# B&R Automation Studio project NAELD004C00R10L518F00 (part 34)

#### Local.var
```iecst
(*2020-03-16*)
(**)
(*Local Action, State & Status*)
VAR
	eAct : eLifterAction := LifterActIdle;
	eStat : eLifterAction := LifterActIdle;
	eMainStatus : eFBStatus := Idle;
	eStatus : eFBStatus := Idle;
	eStatus1 : eFBStatus := Idle;
	eStatus2 : eFBStatus := Idle;
	eStatus3 : eFBStatus := Idle;
	udiStatus : UDINT := 0;
	udiStatus1 : UDINT := 0;
	udiStatus2 : UDINT := 0;
	udiStatus3 : UDINT := 0;
	sStatTxt : STRING[200] := '';
	a_sStatText : ARRAY[0..50] OF STRING[200] := ['Idling','Going A Position','Going B Position','Going C Position','Going D Position','Going E Position','Going F Position','Going G Position','Going H Position','Going A Slot Position','Going Next A Slot Position','Going Previous A Slot Position','Going B Slot Position','Going Next B Slot Position','Going Previous B Slot Position','Going C Slot Position','Going Next C Slot Position','Going Previous C Slot Position','Going D Slot Position','Going Next D Slot Position','Going Previous D Slot Position','Full Homing','Powering On','Powering Off','Homing','Moving Absolute','Moving Relative','Jogging Up','Jogging Down','Jogging Stop','Resetting Axis Error','Stopping','Writing SDO','Background Starting Module OK Check','Background Stopping Module OK Check','Full Moving Relative','Reset Servo Module Node',14('')];
END_VAR
(**)
(*Local Alarm*)
VAR
	tyAlmData : tyAlmDat;
	tyAlmData1 : tyAlmDat;
	tyAlmData2 : tyAlmDat;
	tyAlmData3 : tyAlmDat;
	a_tyAlmText : ARRAY[10000..10299] OF tyAlmTxt := [(sAlmText:='Axis Move Abnormally By External Force',sRcyText:='Servo Motor Abnormal Operation. Reset And Resume Operation. If The Problem Persists, Please Contact Nutek For A Possible Solution.'),(sAlmText:='CANOpen Communication Error, ModuleOK Not TRUE',sRcyText:='Fail While Read/Write Data. Reset The Error And Resume Operation.'),(sAlmText:='Power On Time Out While Going A Position',sRcyText:='Timeout Expired Before Operation Completed. Reset And Resume Operation.'),(sAlmText:='Homing Time Out While Going A Position',sRcyText:='Timeout Expired Before Operation Completed. Reset And Resume Operation.'),(sAlmText:='Move Absolute Time Out While Going A Position',sRcyText:='Timeout Expired Before Operation Completed. Reset And Resume Operation.'),(sAlmText:='Stop Motion Time Out While Going A Position',sRcyText:='Timeout Expired Before Operation Completed. Reset And Resume Operation.'),(sAlmText:='Axis Error Reset Failed While Going A Position',sRcyText:='Axis Error Reset Failed. Please Retry Again Reset Operation. If The Problem Persists, Please Contact Nutek For A Possible Solution.'),(sAlmText:='Axis Error Occur In Move Absolute While Going A Position',sRcyText:='Servo Motor Abnormal Operation. Reset And Resume Operation. If The Problem Persists, Please Contact Nutek For A Possible Solution.'),(sAlmText:='Axis Error Occur In Homing While Going A Position',sRcyText:='Servo Motor Abnormal Operation. Reset And Resume Operation. If The Problem Persists, Please Contact Nutek For A Possible Solution.'),(sAlmText:='Homing Done But Home Flag Is Not Activated While Going A Position',sRcyText:='Servo Motor Abnormal Operation. Reset And Resume Operation. If The Problem Persists, Please Contact Nutek For A Possible Solution.'),(sAlmText:='Forward Limit Activated In Homing While Going A Position',sRcyText:='Forward Limit Switch Is Activated. Reset The Error By Operate The Motor Backwards.'),(sAlmText:='Reverse Limit Activated In Homing While Going A Position',sRcyText:='Reverse Limit Switch Is Activated. Reset The Error By Operate The Motor Backwards.'),(sAlmText:='Forward Limit Activated In Move Absolute While Going A Position',sRcyText:='Forward Limit Switch Is Activated. Reset The Error By Operate The Motor Backwards.'),(sAlmText:='Reverse Limit Activated In Move Absolute While Going A Position',sRcyText:='Reverse Limit Switch Is Activated. Reset The Error By Operate The Motor Backwards.'),(sAlmText:='Power On Time Out While Full Homing',sRcyText:='Timeout Expired Before Operation Completed. Reset And Resume Operation.'),(sAlmText:='Homing Time Out While Full Homing',sRcyText:='Timeout Expired Before Operation Completed. Reset And Resume Operation.'),(sAlmText:='Stop Motion Time Out While Full Homing',sRcyText:='Timeout Expired Before Operation Completed. Reset And Resume Operation.'),(sAlmText:='Axis Error Reset Failed While Full Homing',sRcyText:='Axis Error Reset Failed. Please Retry Again Reset Operation. If The Problem Persists, Please Contact Nutek For A Possible Solution.'),(sAlmText:='Axis Error Occur In Homing While Full Homing',sRcyText:='Servo Motor Abnormal Operation. Reset And Resume Operation. If The Problem Persists, Please Contact Nutek For A Possible Solution.'),(sAlmText:='Homing Done But Home Flag Is Not Activated While Full Homing',sRcyText:='Servo Motor Abnormal Operation. Reset And Resume Operation. If The Problem Persists, Please Contact Nutek For A Possible Solution.'),(sAlmText:='Forward Limit Activated In Homing While Full Homing',sRcyText:='Forward Limit Switch Is Activated. Reset The Error By Operate The Motor Backwards.'),(sAlmText:='Reverse Limit Activated In Homing While Full Homing',sRcyText:='Reverse Limit Switch Is Activated. Reset The Error By Operate The Motor Backwards.'),(sAlmText:='Power On Time Out',sRcyText:='Timeout Expired Before Operation Completed. Reset And Resume Operation.'),(sAlmText:='Power Off Time Out',sRcyText:='Timeout Expired Before Operation Completed. Reset And Resume Operation.'),(sAlmText:='Homing Time Out',sRcyText:='Timeout Expired Before Operation Completed. Reset And Resume Operation.'),(sAlmText:='Move Absolute Time Out',sRcyText:='Timeout Expired Before Operation Completed. Reset And Resume Operation.'),(sAlmText:='Move Relative Time Out',sRcyText:='Timeout Expired Before Operation Completed. Reset And Resume Operation.'),(sAlmText:='Stop Motion Time Out',sRcyText:='Timeout Expired Before Operation Completed. Reset And Resume Operation.'),(sAlmText:='SDO Write Error',sRcyText:='Fail While Write Data. Reset The Error And Resume Operation.'),(sAlmText:='Power On Time Out While Going B Position',sRcyText:='Timeout Expired Before Operation Completed. Reset And Resume Operation.'),(sAlmText:='Homing Time Out While Going B Position',sRcyText:='Timeout Expired Before Operation Completed. Reset And Resume Operation.'),(sAlmText:='Move Absolute Time Out While Going B Position',sRcyText:='Timeout Expired Before Operation Completed. Reset And Resume Operation.'),(sAlmText:='Stop Motion Time Out While Going B Position',sRcyText:='Timeout Expired Before Operation Completed. Reset And Resume Operation.'),(sAlmText:='Axis Error Reset Failed While Going B Position',sRcyText:='Axis Error Reset Failed. Please Retry Again Reset Operation. If The Problem Persists, Please Contact Nutek For A Possible Solution.'),(sAlmText:='Axis Error Occur In Move Absolute While Going B Position',sRcyText:='Servo Motor Abnormal Operation. Reset And Resume Operation. If The Problem Persists, Please Contact Nutek For A Possible Solution.'),(sAlmText:='Axis Error Occur In Homing While Going B Position',sRcyText:='Servo Motor Abnormal Operation. Reset And Resume Operation. If The Problem Persists, Please Contact Nutek For A Possible Solution.'),(sAlmText:='Homing Done But Home Flag Is Not Activated While Going B Position',sRcyText:='Servo Motor Abnormal Operation. Reset And Resume Operation. If The Problem Persists, Please Contact Nutek For A Possible Solution.'),(sAlmText:='Forward Limit Activated In Homing While Going B Position',sRcyText:='Forward Limit Switch Is Activated. Reset The Error By Operate The Motor Backwards.'),(sAlmText:='Reverse Limit Activated In Homing While Going B Position',sRcyText:='Reverse Limit Switch Is Activated. Reset The Error By Operate The Motor Backwards.'),(sAlmText:='Forward Limit Activated In Move Absolute While Going B Position',sRcyText:='Forward Limit Switch Is Activated. Reset The Error By Operate The Motor Backwards.'),(sAlmText:='Reverse Limit Activated In Move Absolute While Going B Position',sRcyText:='Reverse Limit Switch Is Activated. Reset The Error By Operate The Motor Backwards.'),(sAlmText:='Power On Time Out While Going New A Slot Position',sRcyText:='Timeout Expired Before Operation Completed. Reset And Resume Operation.'),(sAlmText:='Homing Time Out While Going New A Slot Position',sRcyText:='Timeout Expired Before Operation Completed. Reset And Resume Operation.'),(sAlmText:='Move Absolute Time Out While Going New A Slot Position',sRcyText:='Timeout Expired Before Operation Completed. Reset And Resume Operation.'),(sAlmText:='Stop Motion Time Out While Going New A Slot Position',sRcyText:='Timeout Expired Before Operation Completed. Reset And Resume Operation.'),(sAlmText:='Axis Error Reset Failed While Going New A Slot Position',sRcyText:='Axis Error Reset Failed. Please Retry Again Reset Operation. If The Problem Persists, Please Contact Nutek For A Possible Solution.'),(sAlmText:='Axis Error Occur In Move Absolute While Going New A Slot Position',sRcyText:='Servo Motor Abnormal Operation. Reset And Resume Operation. If The Problem Persists, Please Contact Nutek For A Possible Solution.'),(sAlmText:='Axis Error Occur In Homing While Going New A Slot Position',sRcyText:='Servo Motor Abnormal Operation. Reset And Resume Operation. If The Problem Persists, Please Contact Nutek For A Possible Solution.'),(sAlmText:='Homing Done But Home Flag Is Not Activated While Going New A Slot Position',sRcyText:='Servo Motor Abnormal Operation. Reset And Resume Operation. If The Problem Persists, Please Contact Nutek For A Possible Solution.'),(sAlmText:='Forward Limit Activated In Homing While Going New A Slot Position',sRcyText:='Forward Limit Switch Is Activated. Reset The Error By Operate The Motor Backwards.'),(sAlmText:='Reverse Limit Activated In Homing While Going New A Slot Position',sRcyText:='Reverse Limit Switch Is Activated. Reset The Error By Operate The Motor Backwards.'),(sAlmText:='Forward Limit Activated In Move Absolute While Going New A Slot Position',sRcyText:='Forward Limit Switch Is Activated. Reset The Error By Operate The Motor Backwards.'),(sAlmText:='Reverse Limit Activated In Move Absolute While Going New A Slot Position',sRcyText:='Reverse Limit Switch Is Activated. Reset The Error By Operate The Motor Backwards.'),(sAlmText:='Power On Time Out While Going Next A Slot Position',sRcyText:='Timeout Expired Before Operation Completed. Reset And Resume Operation.'),(sAlmText:='Homing Time Out While Going Next A Slot Position',sRcyText:='Timeout Expired Before Operation Completed. Reset And Resume Operation.'),(sAlmText:='Move Absolute Time Out While Going Next A Slot Position',sRcyText:='Timeout Expired Before Operation Completed. Reset And Resume Operation.'),(sAlmText:='Stop Motion Time Out While Going Next A Slot Position',sRcyText:='Timeout Expired Before Operation Completed. Reset And Resume Operation.'),(sAlmText:='Axis Error Reset Failed While Going Next A Slot Position',sRcyText:='Axis Error Reset Failed. Please Retry Again Reset Operation. If The Problem Persists, Please Contact Nutek For A Possible Solution.'),(sAlmText:='Axis Error Occur In Move Absolute While Going Next A Slot Position',sRcyText:='Servo Motor Abnormal Operation. Reset And Resume Operation. If The Problem Persists, Please Contact Nutek For A Possible Solution.'),(sAlmText:='Axis Error Occur In Homing While Going Next A Slot Position',sRcyText:='Servo Motor Abnormal Operation. Reset And Resume Operation. If The Problem Persists, Please Contact Nutek For A Possible Solution.'),(sAlmText:='Homing Done But Home Flag Is Not Activated While Going Next A Slot Position',sRcyText:='Servo Motor Abnormal Operation. Reset And Resume Operation. If The Problem Persists, Please Contact Nutek For A Possible Solution.'),(sAlmText:='Forward Limit Activated In Homing While Going Next A Slot Position',sRcyText:='Forward Limit Switch Is Activated. Reset The Error By Operate The Motor Backwards.'),(sAlmText:='Reverse Limit Activated In Homing While Going Next A Slot Position',sRcyText:='Reverse Limit Switch Is Activated. Reset The Error By Operate The Motor Backwards.'),(sAlmText:='Forward Limit Activated In Move Absolute While Going Next A Slot Position',sRcyText:='Forward Limit Switch Is Activated. Reset The Error By Operate The Motor Backwards.'),(sAlmText:='Reverse Limit Activated In Move Absolute While Going Next A Slot Position',sRcyText:='Reverse Limit Switch Is Activated. Reset The Error By Operate The Motor Backwards.'),(sAlmText:='Power On Time Out While Going Previous A Slot Position',sRcyText:='Timeout Expired Before Operation Completed. Reset And Resume Operation.'),(sAlmText:='Homing Time Out While Going Previous A Slot Position',sRcyText:='Timeout Expired Before Operation Completed. Reset And Resume Operation.'),(sAlmText:='Move Absolute Time Out While Going Previous A Slot Position',sRcyText:='Timeout Expired Before Operation Completed. Reset And Resume Operation.'),(sAlmText:='Stop Motion Time Out While Going Previous A Slot Position',sRcyText:='Timeout Expired Before Operation Completed. Reset And Resume Operation.'),(sAlmText:='Axis Error Reset Failed While Going Previous A Slot Position',sRcyText:='Axis Error Reset Failed. Please Retry Again Reset Operation. If The Problem Persists, Please Contact Nutek For A Possible Solution.'),(sAlmText:='Axis Error Occur In Move Absolute While Going Previous A Slot Position',sRcyText:='Servo Motor Abnormal Operation. Reset And Resume Operation. If The Problem Persists, Please Contact Nutek For A Possible Solution.'),(sAlmText:='Axis Error Occur In Homing While Going Previous A Slot Position',sRcyText:='Servo Motor Abnormal Operation. Reset And Resume Operation. If The Problem Persists, Please Contact Nutek For A Possible Solution.'),(sAlmText:='Homing Done But Home Flag Is Not Activated While Going Previous A Slot Position',sRcyText:='Servo Motor Abnormal Operation. Reset And Resume Operation. If The Problem Persists, Please Contact Nutek For A Possible Solution.'),(sAlmText:='Forward Limit Activated In Homing While Going Previous A Slot Position',sRcyText:='Forward Limit Switch Is Activated. Reset The Error By Operate The Motor Backwards.'),(sAlmText:='Reverse Limit Activated In Homing While Going Previous A Slot Position',sRcyText:='Reverse Limit Switch Is Activated. Reset The Error By Operate The Motor Backwards.'),(sAlmText:='Forward Limit Activated In Move Absolute While Going Previous A Slot Position',sRcyText:='Forward Limit Switch Is Activated. Reset The Error By Operate The Motor Backwards.'),(sAlmText:='Reverse Limit Activated In Move Absolute While Going Previous A Slot Position',sRcyText:='Reverse Limit Switch Is Activated. Reset The Error By Operate The Motor Backwards.'),(sAlmText:='Request Absolute Position Out Of Range',sRcyText:='Request Absolute Position Does Not Fall Within The Expected Range.'),(sAlmText:='Power On Time Out While Going C Position',sRcyText:='Timeout Expired Before Operation Completed. Reset And Resume Operation.'),(sAlmText:='Homing Time Out While Going C Position',sRcyText:='Timeout Expired Before Operation Completed. Reset And Resume Operation.'),(sAlmText:='Move Absolute Time Out While Going C Position',sRcyText:='Timeout Expired Before Operation Completed. Reset And Resume Operation.'),(sAlmText:='Stop Motion Time Out While Going C Position',sRcyText:='Timeout Expired Before Operation Completed. Reset And Resume Operation.'),(sAlmText:='Axis Error Reset Failed While Going C Position',sRcyText:='Axis Error Reset Failed. Please Retry Again Reset Operation. If The Problem Persists, Please Contact Nutek For A Possible Solution.'),(sAlmText:='Axis Error Occur In Move Absolute While Going C Position',sRcyText:='Servo Motor Abnormal Operation. Reset And Resume Operation. If The Problem Persists, Please Contact Nutek For A Possible Solution.'),(sAlmText:='Axis Error Occur In Homing While Going C Position',sRcyText:='Servo Motor Abnormal Operation. Reset And Resume Operation. If The Problem Persists, Please Contact Nutek For A Possible Solution.'),(sAlmText:='Homing Done But Home Flag Is Not Activated While Going C Position',sRcyText:='Servo Motor Abnormal Operation. Reset And Resume Operation. If The Problem Persists, Please Contact Nutek For A Possible Solution.'),(sAlmText:='Forward Limit Activated In Homing While Going C Position',sRcyText:='Forward Limit Switch Is Activated. Reset The Error By Operate The Motor Backwards.'),(sAlmText:='Reverse Limit Activated In Homing While Going C Position',sRcyText:='Reverse Limit Switch Is Activated. Reset The Error By Operate The Motor Backwards.'),(sAlmText:='Forward Limit Activated In Move Absolute While Going C Position',sRcyText:='Forward Limit Switch Is Activated. Reset The Error By Operate The Motor Backwards.'),(sAlmText:='Reverse Limit Activated In Move Absolute While Going C Position',sRcyText:='Reverse Limit Switch Is Activated. Reset The Error By Operate The Motor Backwards.'),(sAlmText:='Power On Time Out While Going D Position',sRcyText:='Timeout Expired Before Operation Completed. Reset And Resume Operation.'),(sAlmText:='Homing Time Out While Going D Position',sRcyText:='Timeout Expired Before Operation Completed. Reset And Resume Operation.'),(sAlmText:='Move Absolute Time Out While Going D Position',sRcyText:='Timeout Expired Before Operation Completed. Reset And Resume Operation.'),(sAlmText:='Stop Motion Time Out While Going D Position',sRcyText:='Timeout Expired Before Operation Completed. Reset And Resume Operation.'),(sAlmText:='Axis Error Reset Failed While Going D Position',sRcyText:='Axis Error Reset Failed. Please Retry Again Reset Operation. If The Problem Persists, Please Contact Nutek For A Possible Solution.'),(sAlmText:='Axis Error Occur In Move Absolute While Going D Position',sRcyText:='Servo Motor Abnormal Operation. Reset And Resume Operation. If The Problem Persists, Please Contact Nutek For A Possible Solution.'),(sAlmText:='Axis Error Occur In Homing While Going D Position',sRcyText:='Servo Motor Abnormal Operation. Reset And Resume Operation. If The Problem Persists, Please Contact Nutek For A Possible Solution.'),(sAlmText:='Homing Done But Home Flag Is Not Activated While Going D Position',sRcyText:='Servo Motor Abnormal Operation. Reset And Resume Operation. If The Problem Persists, Please Contact Nutek For A Possible Solution.'),(sAlmText:='Forward Limit Activated In Homing While Going D Position',sRcyText:='Forward Limit Switch Is Activated. Reset The Error By Operate The Motor Backwards.'),(sAlmText:='Reverse Limit Activated In Homing While Going D Position',sRcyText:='Reverse Limit Switch Is Activated. Reset The Error By Operate The Motor Backwards.'),(sAlmText:='Forward Limit Activated In Move Absolute While Going D Position',sRcyText:='Forward Limit Switch Is Activated. Reset The Error By Operate The Motor Backwards.'),(sAlmText:='Reverse Limit Activated In Move Absolute While Going D Position',sRcyText:='Reverse Limit Switch Is Activated. Reset The Error By Operate The Motor Backwards.'),(sAlmText:='Power On Time Out While Going E Position',sRcyText:='Timeout Expired Before Operation Completed. Reset And Resume Operation.'),(sAlmText:='Homing Time Out While Going E Position',sRcyText:='Timeout Expired Before Operation Completed. Reset And Resume Operation.'),(sAlmText:='Move Absolute Time Out While Going E Position',sRcyText:='Timeout Expired Before Operation Completed. Reset And Resume Operation.'),(sAlmText:='Stop Motion Time Out While Going E Position',sRcyText:='Timeout Expired Before Operation Completed. Reset And Resume Operation.'),(sAlmText:='Axis Error Reset Failed While Going E Position',sRcyText:='Axis Error Reset Failed. Please Retry Again Reset Operation. If The Problem Persists, Please Contact Nutek For A Possible Solution.'),(sAlmText:='Axis Error Occur In Move Absolute While Going E Position',sRcyText:='Servo Motor Abnormal Operation. Reset And Resume Operation. If The Problem Persists, Please Contact Nutek For A Possible Solution.'),(sAlmText:='Axis Error Occur In Homing While Going E Position',sRcyText:='Servo Motor Abnormal Operation. Reset And Resume Operation. If The Problem Persists, Please Contact Nutek For A Possible Solution.'),(sAlmText:='Homing Done But Home Flag Is Not Activated While Going E Position',sRcyText:='Servo Motor Abnormal Operation. Reset And Resume Operation. If The Problem Persists, Please Contact Nutek For A Possible Solution.'),(sAlmText:='Forward Limit Activated In Homing While Going E Position',sRcyText:='Forward Limit Switch Is Activated. Reset The Error By Operate The Motor Backwards.'),(sAlmText:='Reverse Limit Activated In Homing While Going E Position',sRcyText:='Reverse Limit Switch Is Activated. Reset The Error By Operate The Motor Backwards.'),(sAlmText:='Forward Limit Activated In Move Absolute While Going E Position',sRcyText:='Forward Limit Switch Is Activated. Reset The Error By Operate The Motor Backwards.'),(sAlmText:='Reverse Limit Activated In Move Absolute While Going E Position',sRcyText:='Reverse Limit Switch Is Activated. Reset The Error By Operate The Motor Backwards.'),(sAlmText:='Power On Time Out While Going F Position',sRcyText:='Timeout Expired Before Operation Completed. Reset And Resume Operation.'),(sAlmText:='Homing Time Out While Going F Position',sRcyText:='Timeout Expired Before Operation Completed. Reset And Resume Operation.'),(sAlmText:='Move Absolute Time Out While Going F Position',sRcyText:='Timeout Expired Before Operation Completed. Reset And Resume Operation.'),(sAlmText:='Stop Motion Time Out While Going F Position',sRcyText:='Timeout Expired Before Operation Completed. Reset And Resume Operation.'),(sAlmText:='Axis Error Reset Failed While Going F Position',sRcyText:='Axis Error Reset Failed. Please Retry Again Reset Operation. If The Problem Persists, Please Contact Nutek For A Possible Solution.'),(sAlmText:='Axis Error Occur In Move Absolute While Going F Position',sRcyText:='Servo Motor Abnormal Operation. Reset And Resume Operation. If The Problem Persists, Please Contact Nutek For A Possible Solution.'),(sAlmText:='Axis Error Occur In Homing While Going F Position',sRcyText:='Servo Motor Abnormal Operation. Reset And Resume Operation. If The Problem Persists, Please Contact Nutek For A Possible Solution.'),(sAlmText:='Homing Done But Home Flag Is Not Activated While Going F Position',sRcyText:='Servo Motor Abnormal Operation. Reset And Resume Operation. If The Problem Persists, Please Contact Nutek For A Possible Solution.'),(sAlmText:='Forward Limit Activated In Homing While Going F Position',sRcyText:='Forward Limit Switch Is Activated. Reset The Error By Operate The Motor Backwards.'),(sAlmText:='Reverse Limit Activated In Homing While Going F Position',sRcyText:='Reverse Limit Switch Is Activated. Reset The Error By Operate The Motor Backwards.'),(sAlmText:='Forward Limit Activated In Move Absolute While Going F Position',sRcyText:='Forward Limit Switch Is Activated. Reset The Error By Operate The Motor Backwards.'),(sAlmText:='Reverse Limit Activated In Move Absolute While Going F Position',sRcyText:='Reverse Limit Switch Is Activated. Reset The Error By Operate The Motor Backwards.'),(sAlmText:='Power On Time Out While Going G Position',sRcyText:='Timeout Expired Before Operation Completed. Reset And Resume Operation.'),(sAlmText:='Homing Time Out While Going G Position',sRcyText:='Timeout Expired Before Operation Completed. Reset And Resume Operation.'),(sAlmText:='Move Absolute Time Out While Going G Position',sRcyText:='Timeout Expired Before Operation Completed. Reset And Resume Operation.'),(sAlmText:='Stop Motion Time Out While Going G Position',sRcyText:='Timeout Expired Before Operation Completed. Reset And Resume Operation.'),(sAlmText:='Axis Error Reset Failed While Going G Position',sRcyText:='Axis Error Reset Failed. Please Retry Again Reset Operation. If The Problem Persists, Please Contact Nutek For A Possible Solution.'),(sAlmText:='Axis Error Occur In Move Absolute While Going G Position',sRcyText:='Servo Motor Abnormal Operation. Reset And Resume Operation. If The Problem Persists, Please Contact Nutek For A Possible Solution.'),(sAlmText:='Axis Error Occur In Homing While Going G Position',sRcyText:='Servo Motor Abnormal Operation. Reset And Resume Operation. If The Problem Persists, Please Contact Nutek For A Possible Solution.'),(sAlmText:='Homing Done But Home Flag Is Not Activated While Going G Position',sRcyText:='Servo Motor Abnormal Operation. Reset And Resume Operation. If The Problem Persists, Please Contact Nutek For A Possible Solution.'),(sAlmText:='Forward Limit Activated In Homing While Going G Position',sRcyText:='Forward Limit Switch Is Activated. Reset The Error By Operate The Motor Backwards.'),(sAlmText:='Reverse Limit Activated In Homing While Going G Position',sRcyText:='Reverse Limit Switch Is Activated. Reset The Error By Operate The Motor Backwards.'),(sAlmText:='Forward Limit Activated In Move Absolute While Going G Position',sRcyText:='Forward Limit Switch Is Activated. Reset The Error By Operate The Motor Backwards.'),(sAlmText:='Reverse Limit Activated In Move Absolute While Going G Position',sRcyText:='Reverse Limit Switch Is Activated. Reset The Error By Operate The Motor Backwards.'),(sAlmText:='Power On Time Out While Going H Position',sRcyText:='Timeout Expired Before Operation Completed. Reset And Resume Operation.'),(sAlmText:='Homing Time Out While Going H Position',sRcyText:='Timeout Expired Before Operation Completed. Reset And Resume Operation.'),(sAlmText:='Move Absolute Time Out While Going H Position',sRcyText:='Timeout Expired Before Operation Completed. Reset And Resume Operation.'),(sAlmText:='Stop Motion Time Out While Going H Position',sRcyText:='Timeout Expired Before Operation Completed. Reset And Resume Operation.'),(sAlmText:='Axis Error Reset Failed While Going H Position',sRcyText:='Axis Error Reset Failed. Please Retry Again Reset Operation. If The Problem Persists, Please Contact Nutek For A Possible Solution.'),(sAlmText:='Axis Error Occur In Move Absolute While Going H Position',sRcyText:='Servo Motor Abnormal Operation. Reset And Resume Operation. If The Problem Persists, Please Contact Nutek For A Possible Solution.'),(sAlmText:='Axis Error Occur In Homing While Going H Position',sRcyText:='Servo Motor Abnormal Operation. Reset And Resume Operation. If The Problem Persists, Please Contact Nutek For A Possible Solution.'),(sAlmText:='Homing Done But Home Flag Is Not Activated While Going H Position',sRcyText:='Servo Motor Abnormal Operation. Reset And Resume Operation. If The Problem Persists, Please Contact Nutek For A Possible Solution.'),(sAlmText:='Forward Limit Activated In Homing While Going H Position',sRcyText:='Forward Limit Switch Is Activated. Reset The Error By Operate The Motor Backwards.'),(sAlmText:='Reverse Limit Activated In Homing While Going H Position',sRcyText:='Reverse Limit Switch Is Activated. Reset The Error By Operate The Motor Backwards.'),(sAlmText:='Forward Limit Activated In Move Absolute While Going H Position',sRcyText:='Forward Limit Switch Is Activated. Reset The Error By Operate The Motor Backwards.'),(sAlmText:='Reverse Limit Activated In Move Absolute While Going H Position',sRcyText:='Reverse Limit Switch Is Activated. Reset The Error By Operate The Motor Backwards.'),(sAlmText:='Power On Time Out While Going New B Slot Position',sRcyText:='Timeout Expired Before Operation Completed. Reset And Resume Operation.'),(sAlmText:='Homing Time Out While Going New B Slot Position',sRcyText:='Timeout Expired Before Operation Completed. Reset And Resume Operation.'),(sAlmText:='Move Absolute Time Out While Going New B Slot Position',sRcyText:='Timeout Expired Before Operation Completed. Reset And Resume Operation.'),(sAlmText:='Stop Motion Time Out While Going New B Slot Position',sRcyText:='Timeout Expired Before Operation Completed. Reset And Resume Operation.'),(sAlmText:='Axis Error Reset Failed While Going New B Slot Position',sRcyText:='Axis Error Reset Failed. Please Retry Again Reset Operation. If The Problem Persists, Please Contact Nutek For A Possible Solution.'),(sAlmText:='Axis Error Occur In Move Absolute While Going New B Slot Position',sRcyText:='Servo Motor Abnormal Operation. Reset And Resume Operation. If The Problem Persists, Please Contact Nutek For A Possible Solution.'),(sAlmText:='Axis Error Occur In Homing While Going New B Slot Position',sRcyText:='Servo Motor Abnormal Operation. Reset And Resume Operation. If The Problem Persists, Please Contact Nutek For A Possible Solution.'),(sAlmText:='Homing Done But Home Flag Is Not Activated While Going New B Slot Position',sRcyText:='Servo Motor Abnormal Operation. Reset And Resume Operation. If The Problem Persists, Please Contact Nutek For A Possible Solution.'),(sAlmText:='Forward Limit Activated In Homing While Going New B Slot Position',sRcyText:='Forward Limit Switch Is Activated. Reset The Error By Operate The Motor Backwards.'),(sAlmText:='Reverse Limit Activated In Homing While Going New B Slot Position',sRcyText:='Reverse Limit Switch Is Activated. Reset The Error By Operate The Motor Backwards.'),(sAlmText:='Forward Limit Activated In Move Absolute While Going New B Slot Position',sRcyText:='Forward Limit Switch Is Activated. Reset The Error By Operate The Motor Backwards.'),(sAlmText:='Reverse Limit Activated In Move Absolute While Going New B Slot Position',sRcyText:='Reverse Limit Switch Is Activated. Reset The Error By Operate The Motor Backwards.'),(sAlmText:='Power On Time Out While Going Next B Slot Position',sRcyText:='Timeout Expired Before Operation Completed. Reset And Resume Operation.'),(sAlmText:='Homing Time Out While Going Next B Slot Position',sRcyText:='Timeout Expired Before Operation Completed. Reset And Resume Operation.'),(sAlmText:='Move Absolute Time Out While Going Next B Slot Position',sRcyText:='Timeout Expired Before Operation Completed. Reset And Resume Operation.'),(sAlmText:='Stop Motion Time Out While Going Next B Slot Position',sRcyText:='Timeout Expired Before Operation Completed. Reset And Resume Operation.'),(sAlmText:='Axis Error Reset Failed While Going Next B Slot Position',sRcyText:='Axis Error Reset Failed. Please Retry Again Reset Operation. If The Problem Persists, Please Contact Nutek For A Possible Solution.'),(sAlmText:='Axis Error Occur In Move Absolute While Going Next B Slot Position',sRcyText:='Servo Motor Abnormal Operation. Reset And Resume Operation. If The Problem Persists, Please Contact Nutek For A Possible Solution.'),(sAlmText:='Axis Error Occur In Homing While Going Next B Slot Position',sRcyText:='Servo Motor Abnormal Operation. Reset And Resume Operation. If The Problem Persists, Please Contact Nutek For A Possible Solution.'),(sAlmText:='Homing Done But Home Flag Is Not Activated While Going Next B Slot Position',sRcyText:='Servo Motor Abnormal Operation. Reset And Resume Operation. If The Problem Persists, Please Contact Nutek For A Possible Solution.'),(sAlmText:='Forward Limit Activated In Homing While Going Next B Slot Position',sRcyText:='Forward Limit Switch Is Activated. Reset The Error By Operate The Motor Backwards.'),(sAlmText:='Reverse Limit Activated In Homing While Going Next B Slot Position',sRcyText:='Reverse Limit Switch Is Activated. Reset The Error By Operate The Motor Backwards.'),(sAlmText:='Forward Limit Activated In Move Absolute While Going Next B Slot Position',sRcyText:='Forward Limit Switch Is Activated. Reset The Error By Operate The Motor Backwards.'),(sAlmText:='Reverse Limit Activated In Move Absolute While Going Next B Slot Position',sRcyText:='Reverse Limit Switch Is Activated. Reset The Error By Operate The Motor Backwards.'),(sAlmText:='Power On Time Out While Going Previous B Slot Position',sRcyText:='Timeout Expired Before Operation Completed. Reset And Resume Operation.'),(sAlmText:='Homing Time Out While Going Previous B Slot Position',sRcyText:='Timeout Expired Before Operation Completed. Reset And Resume Operation.'),(sAlmText:='Move Absolute Time Out While Going Previous B Slot Position',sRcyText:='Timeout Expired Before Operation Completed. Reset And Resume Operation.'),(sAlmText:='Stop Motion Time Out While Going Previous B Slot Position',sRcyText:='Timeout Expired Before Operation Completed. Reset And Resume Operation.'),(sAlmText:='Axis Error Reset Failed While Going Previous B Slot Position',sRcyText:='Axis Error Reset Failed. Please Retry Again Reset Operation. If The Problem Persists, Please Contact Nutek For A Possible Solution.'),(sAlmText:='Axis Error Occur In Move Absolute While Going Previous B Slot Position',sRcyText:='Servo Motor Abnormal Operation. Reset And Resume Operation. If The Problem Persists, Please Contact Nutek For A Possible Solution.'),(sAlmText:='Axis Error Occur In Homing While Going Previous B Slot Position',sRcyText:='Servo Motor Abnormal Operation. Reset And Resume Operation. If The Problem Persists, Please Contact Nutek For A Possible Solution.'),(sAlmText:='Homing Done But Home Flag Is Not Activated While Going Previous B Slot Position',sRcyText:='Servo Motor Abnormal Operation. Reset And Resume Operation. If The Problem Persists, Please Contact Nutek For A Possible Solution.'),(sAlmText:='Forward Limit Activated In Homing While Going Previous B Slot Position',sRcyText:='Forward Limit Switch Is Activated. Reset The Error By Operate The Motor Backwards.'),(sAlmText:='Reverse Limit Activated In Homing While Going Previous B Slot Position',sRcyText:='Reverse Limit Switch Is Activated. Reset The Error By Operate The Motor Backwards.'),(sAlmText:='Forward Limit Activated In Move Absolute While Going Previous B Slot Position',sRcyText:='Forward Limit Switch Is Activated. Reset The Error By Operate The Motor Backwards.'),(sAlmText:='Reverse Limit Activated In Move Absolute While Going Previous B Slot Position',sRcyText:='Reverse Limit Switch Is Activated. Reset The Error By Operate The Motor Backwards.'),(sAlmText:='Power On Time Out While Going New C Slot Position',sRcyText:='Timeout Expired Before Operation Completed. Reset And Resume Operation.'),(sAlmText:='Homing Time Out While Going New C Slot Position',sRcyText:='Timeout Expired Before Operation Completed. Reset And Resume Operation.'),(sAlmText:='Move Absolute Time Out While Going New C Slot Position',sRcyText:='Timeout Expired Before Operation Completed. Reset And Resume Operation.'),(sAlmText:='Stop Motion Time Out While Going New C Slot Position',sRcyText:='Timeout Expired Before Operation Completed. Reset And Resume Operation.'),(sAlmText:='Axis Error Reset Failed While Going New C Slot Position',sRcyText:='Axis Error Reset Failed. Please Retry Again Reset Operation. If The Problem Persists, Please Contact Nutek For A Possible Solution.'),(sAlmText:='Axis Error Occur In Move Absolute While Going New C Slot Position',sRcyText:='Servo Motor Abnormal Operation. Reset And Resume Operation. If The Problem Persists, Please Contact Nutek For A Possible Solution.'),(sAlmText:='Axis Error Occur In Homing While Going New C Slot Position',sRcyText:='Servo Motor Abnormal Operation. Reset And Resume Operation. If The Problem Persists, Please Contact Nutek For A Possible Solution.'),(sAlmText:='Homing Done But Home Flag Is Not Activated While Going New C Slot Position',sRcyText:='Servo Motor Abnormal Operation. Reset And Resume Operation. If The Problem Persists, Please Contact Nutek For A Possible Solution.'),(sAlmText:='Forward Limit Activated In Homing While Going New C Slot Position',sRcyText:='Forward Limit Switch Is Activated. Reset The Error By Operate The Motor Backwards.'),(sAlmText:='Reverse Limit Activated In Homing While Going New C Slot Position',sRcyText:='Reverse Limit Switch Is Activated. Reset The Error By Operate The Motor Backwards.'),(sAlmText:='Forward Limit Activated In Move Absolute While Going New C Slot Position',sRcyText:='Forward Limit Switch Is Activated. Reset The Error By Operate The Motor Backwards.'),(sAlmText:='Reverse Limit Activated In Move Absolute While Going New C Slot Position',sRcyText:='Reverse Limit Switch Is Activated. Reset The Error By Operate The Motor Backwards.'),(sAlmText:='Power On Time Out While Going Next C Slot Position',sRcyText:='Timeout Expired Before Operation Completed. Reset And Resume Operation.'),(sAlmText:='Homing Time Out While Going Next C Slot Position',sRcyText:='Timeout Expired Before Operation Completed. Reset And Resume Operation.'),(sAlmText:='Move Absolute Time Out While Going Next C Slot Position',sRcyText:='Timeout Expired Before Operation Completed. Reset And Resume Operation.'),(sAlmText:='Stop Motion Time Out While Going Next C Slot Position',sRcyText:='Timeout Expired Before Operation Completed. Reset And Resume Operation.'),(sAlmText:='Axis Error Reset Failed While Going Next C Slot Position',sRcyText:='Axis Error Reset Failed. Please Retry Again Reset Operation. If The Problem Persists, Please Contact Nutek For A Possible Solution.'),(sAlmText:='Axis Error Occur In Move Absolute While Going Next C Slot Position',sRcyText:='Servo Motor Abnormal Operation. Reset And Resume Operation. If The Problem Persists, Please Contact Nutek For A Possible Solution.'),(sAlmText:='Axis Error Occur In Homing While Going Next C Slot Position',sRcyText:='Servo Motor Abnormal Operation. Reset And Resume Operation. If The Problem Persists, Please Contact Nutek For A Possible Solution.'),(sAlmText:='Homing Done But Home Flag Is Not Activated While Going Next C Slot Position',sRcyText:='Servo Motor Abnormal Operation. Reset And Resume Operation. If The Problem Persists, Please Contact Nutek For A Possible Solution.'),(sAlmText:='Forward Limit Activated In Homing While Going Next C Slot Position',sRcyText:='Forward Limit Switch Is Activated. Reset The Error By Operate The Motor Backwards.'),(sAlmText:='Reverse Limit Activated In Homing While Going Next C Slot Position',sRcyText:='Reverse Limit Switch Is Activated. Reset The Error By Operate The Motor Backwards.'),(sAlmText:='Forward Limit Activated In Move Absolute While Going Next C Slot Position',sRcyText:='Forward Limit Switch Is Activated. Reset The Error By Operate The Motor Backwards.'),(sAlmText:='Reverse Limit Activated In Move Absolute While Going Next C Slot Position',sRcyText:='Reverse Limit Switch Is Activated. Reset The Error By Operate The Motor Backwards.'),(sAlmText:='Power On Time Out While Going Previous C Slot Position',sRcyText:='Timeout Expired Before Operation Completed. Reset And Resume Operation.'),(sAlmText:='Homing Time Out While Going Previous C Slot Position',sRcyText:='Timeout Expired Before Operation Completed. Reset And Resume Operation.'),(sAlmText:='Move Absolute Time Out While Going Previous C Slot Position',sRcyText:='Timeout Expired Before Operation Completed. Reset And Resume Operation.'),(sAlmText:='Stop Motion Time Out While Going Previous C Slot Position',sRcyText:='Timeout Expired Before Operation Completed. Reset And Resume Operation.'),(sAlmText:='Axis Error Reset Failed While Going Previous C Slot Position',sRcyText:='Axis Error Reset Failed. Please Retry Again Reset Operation. If The Problem Persists, Please Contact Nutek For A Possible Solution.'),(sAlmText:='Axis Error Occur In Move Absolute While Going Previous C Slot Position',sRcyText:='Servo Motor Abnormal Operation. Reset And Resume Operation. If The Problem Persists, Please Contact Nutek For A Possible Solution.'),(sAlmText:='Axis Error Occur In Homing While Going Previous C Slot Position',sRcyText:='Servo Motor Abnormal Operation. Reset And Resume Operation. If The Problem Persists, Please Contact Nutek For A Possible Solution.'),(sAlmText:='Homing Done But Home Flag Is Not Activated While Going Previous C Slot Position',sRcyText:='Servo Motor Abnormal Operation. Reset And Resume Operation. If The Problem Persists, Please Contact Nutek For A Possible Solution.'),(sAlmText:='Forward Limit Activated In Homing While Going Previous C Slot Position',sRcyText:='Forward Limit Switch Is Activated. Reset The Error By Operate The Motor Backwards.'),(sAlmText:='Reverse Limit Activated In Homing While Going Previous C Slot Position',sRcyText:='Reverse Limit Switch Is Activated. Reset The Error By Operate The Motor Backwards.'),(sAlmText:='Forward Limit Activated In Move Absolute While Going Previous C Slot Position',sRcyText:='Forward Limit Switch Is Activated. Reset The Error By Operate The Motor Backwards.'),(sAlmText:='Reverse Limit Activated In Move Absolute While Going Previous C Slot Position',sRcyText:='Reverse Limit Switch Is Activated. Reset The Error By Operate The Motor Backwards.'),(sAlmText:='Power On Time Out While Going New D Slot Position',sRcyText:='Timeout Expired Before Operation Completed. Reset And Resume Operation.'),(sAlmText:='Homing Time Out While Going New D Slot Position',sRcyText:='Timeout Expired Before Operation Completed. Reset And Resume Operation.'),(sAlmText:='Move Absolute Time Out While Going New D Slot Position',sRcyText:='Timeout Expired Before Operation Completed. Reset And Resume Operation.'),(sAlmText:='Stop Motion Time Out While Going New D Slot Position',sRcyText:='Timeout Expired Before Operation Completed. Reset And Resume Operation.'),(sAlmText:='Axis Error Reset Failed While Going New D Slot Position',sRcyText:='Axis Error Reset Failed. Please Retry Again Reset Operation. If The Problem Persists, Please Contact Nutek For A Possible Solution.'),(sAlmText:='Axis Error Occur In Move Absolute While Going New D Slot Position',sRcyText:='Servo Motor Abnormal Operation. Reset And Resume Operation. If The Problem Persists, Please Contact Nutek For A Possible Solution.'),(sAlmText:='Axis Error Occur In Homing While Going New D Slot Position',sRcyText:='Servo Motor Abnormal Operation. Reset And Resume Operation. If The Problem Persists, Please Contact Nutek For A Possible Solution.'),(sAlmText:='Homing Done But Home Flag Is Not Activated While Going New D Slot Position',sRcyText:='Servo Motor Abnormal Operation. Reset And Resume Operation. If The Problem Persists, Please Contact Nutek For A Possible Solution.'),(sAlmText:='Forward Limit Activated In Homing While Going New D Slot Position',sRcyText:='Forward Limit Switch Is Activated. Reset The Error By Operate The Motor Backwards.'),(sAlmText:='Reverse Limit Activated In Homing While Going New D Slot Position',sRcyText:='Reverse Limit Switch Is Activated. Reset The Error By Operate The Motor Backwards.'),(sAlmText:='Forward Limit Activated In Move Absolute While Going New D Slot Position',sRcyText:='Forward Limit Switch Is Activated. Reset The Error By Operate The Motor Backwards.'),(sAlmText:='Reverse Limit Activated In Move Absolute While Going New D Slot Position',sRcyText:='Reverse Limit Switch Is Activated. Reset The Error By Operate The Motor Backwards.'),(sAlmText:='Power On Time Out While Going Next D Slot Position',sRcyText:='Timeout Expired Before Operation Completed. Reset And Resume Operation.'),(sAlmText:='Homing Time Out While Going Next D Slot Position',sRcyText:='Timeout Expired Before Operation Completed. Reset And Resume Operation.'),(sAlmText:='Move Absolute Time Out While Going Next D Slot Position',sRcyText:='Timeout Expired Before Operation Completed. Reset And Resume Operation.'),(sAlmText:='Stop Motion Time Out While Going Next D Slot Position',sRcyText:='Timeout Expired Before Operation Completed. Reset And Resume Operation.'),(sAlmText:='Axis Error Reset Failed While Going Next D Slot Position',sRcyText:='Axis Error Reset Failed. Please Retry Again Reset Operation. If The Problem Persists, Please Contact Nutek For A Possible Solution.'),(sAlmText:='Axis Error Occur In Move Absolute While Going Next D Slot Position',sRcyText:='Servo Motor Abnormal Operation. Reset And Resume Operation. If The Problem Persists, Please Contact Nutek For A Possible Solution.'),(sAlmText:='Axis Error Occur In Homing While Going Next D Slot Position',sRcyText:='Servo Motor Abnormal Operation. Reset And Resume Operation. If The Problem Persists, Please Contact Nutek For A Possible Solution.'),(sAlmText:='Homing Done But Home Flag Is Not Activated While Going Next D Slot Position',sRcyText:='Servo Motor Abnormal Operation. Reset And Resume Operation. If The Problem Persists, Please Contact Nutek For A Possible Solution.'),(sAlmText:='Forward Limit Activated In Homing While Going Next D Slot Position',sRcyText:='Forward Limit Switch Is Activated. Reset The Error By Operate The Motor Backwards.'),(sAlmText:='Reverse Limit Activated In Homing While Going Next D Slot Position',sRcyText:='Reverse Limit Switch Is Activated. Reset The Error By Operate The Motor Backwards.'),(sAlmText:='Forward Limit Activated In Move Absolute While Going Next D Slot Position',sRcyText:='Forward Limit Switch Is Activated. Reset The Error By Operate The Motor Backwards.'),(sAlmText:='Reverse Limit Activated In Move Absolute While Going Next D Slot Position',sRcyText:='Reverse Limit Switch Is Activated. Reset The Error By Operate The Motor Backwards.'),(sAlmText:='Power On Time Out While Going Previous D Slot Position',sRcyText:='Timeout Expired Before Operation Completed. Reset And Resume Operation.'),(sAlmText:='Homing Time Out While Going Previous D Slot Position',sRcyText:='Timeout Expired Before Operation Completed. Reset And Resume Operation.'),(sAlmText:='Move Absolute Time Out While Going Previous D Slot Position',sRcyText:='Timeout Expired Before Operation Completed. Reset And Resume Operation.'),(sAlmText:='Stop Motion Time Out While Going Previous D Slot Position',sRcyText:='Timeout Expired Before Operation Completed. Reset And Resume Operation.'),(sAlmText:='Axis Error Reset Failed While Going Previous D Slot Position',sRcyText:='Axis Error Reset Failed. Please Retry Again Reset Operation. If The Problem Persists, Please Contact Nutek For A Possible Solution.'),(sAlmText:='Axis Error Occur In Move Absolute While Going Previous D Slot Position',sRcyText:='Servo Motor Abnormal Operation. Reset And Resume Operation. If The Problem Persists, Please Contact Nutek For A Possible Solution.'),(sAlmText:='Axis Error Occur In Homing While Going Previous D Slot Position',sRcyText:='Servo Motor Abnormal Operation. Reset And Resume Operation. If The Problem Persists, Please Contact Nutek For A Possible Solution.'),(sAlmText:='Homing Done But Home Flag Is Not Activated While Going Previous D Slot Position',sRcyText:='Servo Motor Abnormal Operation. Reset And Resume Operation. If The Problem Persists, Please Contact Nutek For A Possible Solution.'),(sAlmText:='Forward Limit Activated In Homing While Going Previous D Slot Position',sRcyText:='Forward Limit Switch Is Activated. Reset The Error By Operate The Motor Backwards.'),(sAlmText:='Reverse Limit Activated In Homing While Going Previous D Slot Position',sRcyText:='Reverse Limit Switch Is Activated. Reset The Error By Operate The Motor Backwards.'),(sAlmText:='Forward Limit Activated In Move Absolute While Going Previous D Slot Position',sRcyText:='Forward Limit Switch Is Activated. Reset The Error By Operate The Motor Backwards.'),(sAlmText:='Reverse Limit Activated In Move Absolute While Going Previous D Slot Position',sRcyText:='Reverse Limit Switch Is Activated. Reset The Error By Operate The Motor Backwards.'),(sAlmText:='Sensor Interrupt Lifter Movement',sRcyText:='Operation Stop Due To The Interruption Of Sensor While Lifter Moving. Solve The Interruption To Resume Operation.'),(sAlmText:='Power On Time Out While Full Moving Relative',sRcyText:='Timeout Expired Before Operation Completed. Reset And Resume Operation.'),(sAlmText:='Move Relative Time Out Full Moving Relative',sRcyText:='Timeout Expired Before Operation Completed. Reset And Resume Operation.'),(sAlmText:='Stop Motion Time Out While Full Moving Relative',sRcyText:='Timeout Expired Before Operation Completed. Reset And Resume Operation.'),(sAlmText:='Axis Error Reset Failed While Full Moving Relative',sRcyText:='Axis Error Reset Failed. Please Retry Again Reset Operation. If The Problem Persists, Please Contact Nutek For A Possible Solution.'),37((0))];
END_VAR
(**)
(*Local Output*)
VAR
	tyParamOut : tyMotionCANParamOut;
	sAxisErrTxt : STRING[80];
	bSltAPosDiff : BOOL;
	bSltBPosDiff : BOOL;
	bSltCPosDiff : BOOL;
	bSltDPosDiff : BOOL;
	diCurrSltA : DINT;
	diCurrSltB : DINT;
	diCurrSltC : DINT;
	diCurrSltD : DINT;
	bAPosDiff : BOOL;
	bBPosDiff : BOOL;
	bCPosDiff : BOOL;
	bDPosDiff : BOOL;
	bEPosDiff : BOOL;
	bFPosDiff : BOOL;
	bGPosDiff : BOOL;
	bHPosDiff : BOOL;
	bJogging : BOOL;
	bUpSen : BOOL;
	bDownSen : BOOL;
END_VAR
(**)
(*Local Input*)
VAR
	udiRstErr : UDINT := 0;
	bPrep : BOOL := TRUE;
	bEn : BOOL := TRUE;
	bDis : BOOL := FALSE;
	bOps : BOOL := FALSE;
	bManual : BOOL := FALSE;
	diGoASlt : DINT := 1;
	diASltToSltDist : DINT := 10000;
	diASlt1Pos : DINT := 500000;
	diGoBSlt : DINT := 1;
	diBSltToSltDist : DINT := 10000;
	diBSlt1Pos : DINT := 500000;
	diGoCSlt : DINT := 1;
	diCSltToSltDist : DINT := 10000;
	diCSlt1Pos : DINT := 500000;
	diGoDSlt : DINT := 1;
	diDSltToSltDist : DINT := 10000;
	diDSlt1Pos : DINT := 500000;
	diAPos : DINT := 0;
	diBPos : DINT := 0;
	diCPos : DINT := 0;
	diDPos : DINT := 0;
	diEPos : DINT := 0;
	diFPos : DINT := 0;
	diGPos : DINT := 0;
	diHPos : DINT := 0;
	tyTuning : tyMotionCANTuning;
	diJogVelInUMPS : DINT := 50000;
	diMovePosInUM : DINT := 0;
	diMoveDistInUM : DINT := 0;
	diMoveVelInUMPS : DINT := 50000;
	diMoveAcc : DINT := 500;
	diMoveDec : DINT := 500;
	diMinAbsPosInUM : DINT := -10000;
	diMaxAbsPosInUM : DINT := 10000000;
	bInterruptSensor1 : BOOL;
	bInterruptSensor2 : BOOL;
	bInterruptSensor3 : BOOL;
	bInterruptSensor4 : BOOL;
	bInterruptSensor5 : BOOL;
	bInterruptSensor6 : BOOL;
	bDir : BOOL;
	bNoIndexPulse : BOOL;
	usiNode : USINT;
	sDevice : STRING[3];
	sProgNm : STRING[15] := 'LifterBtm';
	tyParamInHm : tyMotionCANParamInHm;
	tyParamInConvert : tyMotionCANParamInConvert;
	bNtSettingsLoadDone : BOOL := TRUE;
END_VAR
(**)
(*Local*)
VAR
	bRstErr : BOOL;
	udiRstErrOld : UDINT;
	bInitDone : BOOL;
	bInitialDone : BOOL;
	bModuleOKChk : BOOL := FALSE;
	bModuleOK : BOOL;
	bModuleNotOK : BOOL := TRUE;
	bModuleNotOKLock : BOOL;
	bNotInterruptible : BOOL;
	diExpectSlt : DINT;
	diExpectPosInUM : DINT;
	diActualPosInUMOld : DINT;
	usiRstStep : USINT := 0;
	usiStep : USINT;
	usiCount : USINT;
	fbTm : TON := (PT:=T#2s);
	fbServoModuleNotOk : TON := (IN:=FALSE,PT:=T#2s);
	fbServoModuleOk : TON := (IN:=FALSE,PT:=T#5s);
	fbRstNodeTimer : TON := (PT:=T#3s);
	tyParamInMove : tyMotionCANParamInMove;
	tyParamInDriver : tyMotionCANDriverIn := (siModOfOptDisp_6061:=6);
	tyParamOutDriver : tyMotionCANDriverOut;
	fbStop : fbMotionCANStop;
	fbRstAxisErr : fbMotionCANRstAxisErr;
	fbJog : fbMotionCANJog;
	fbMovRel : fbMotionCANMovRel;
	fbMovAbs : fbMotionCANMovAbs;
	fbHoming : fbMotionCANHoming;
	fbPwrOff : fbMotionCANPwrOff;
	fbPwrOn : fbMotionCANPwrOn;
	fbFullHm : fbMotionCANFullHm;
	fbFullMovRel : fbMotionCANFullMovRel;
	fbFullMovAbs : fbMotionCANFullMovAbs;
	fbModuleOK : fbMotionCANModuleOK;
	fbSDOWrite : fbCANSDOWriteArrayParam;
	bInletShutterCloseRS : BOOL;
	udiModuleNum : UDINT := 1201;
END_VAR
```

#### Act_Alarm1.st
```iecst
(** 2020-03-16 **)
ACTION Act_Alarm1:

	//Error
	IF EDGEPOS(eStatus1 = Error) THEN

		tyAlmData1.sProgNm		:= p_sProgNm;
		tyAlmData1.udiCode		:= udiStatus1;
		tyAlmData1.eSeverity	:= AlmSeverityError;
		tyAlmData1.udiRunTime	:= tyAlmData1.udiRunTime + 1;
		tyAlmData1.bAlm			:= TRUE;
		tyAlmData1.udiModuleNum  := udiModuleNum;
		g_sLifterBtmProgNm		:= p_sProgNm;

		//Get Error Message
		IF tyAlmData1.udiCode < 10000 OR tyAlmData1.udiCode > 10299 THEN
			tyAlmData1.sAlmMsg	:= 'Unknown';
			tyAlmData1.sRcyMsg	:= 'Unknown';
		ELSE
			tyAlmData1.sAlmMsg	:= a_tyAlmText[tyAlmData1.udiCode].sAlmText;
			tyAlmData1.sRcyMsg	:= a_tyAlmText[tyAlmData1.udiCode].sRcyText;
		END_IF

		sStatTxt	:= tyAlmData1.sAlmMsg;

	ELSIF bRstErr AND (tyAlmData1.udiCode <> 0) THEN

		tyAlmData1.udiCode		:= 0;
		tyAlmData1.eSeverity	:= AlmSeverityNA;
		tyAlmData1.sAlmMsg		:= '';
		tyAlmData1.sRcyMsg		:= '';
		tyAlmData1.bAlm			:= FALSE;
		sStatTxt	:= a_sStatText[eStat];

	END_IF

END_ACTION
```

#### Act_Alarm2.st
```iecst
(** 2020-03-16 **)
ACTION Act_Alarm2:

	//Error
	IF EDGEPOS(eStatus2 = Error) THEN

		tyAlmData2.sProgNm		:= p_sProgNm;
		tyAlmData2.udiCode		:= udiStatus2;
		tyAlmData2.eSeverity	:= AlmSeverityError;
		tyAlmData2.udiRunTime	:= tyAlmData2.udiRunTime + 1;
		tyAlmData2.bAlm			:= TRUE;
		tyAlmData2.udiModuleNum  := udiModuleNum;
		g_sLifterBtmProgNm		:= p_sProgNm;
		//Get Error Message
		IF tyAlmData2.udiCode < 10000 OR tyAlmData2.udiCode > 10299 THEN
			tyAlmData2.sAlmMsg	:= 'Unknown';
			tyAlmData2.sRcyMsg	:= 'Unknown';
		ELSE
			tyAlmData2.sAlmMsg	:= a_tyAlmText[tyAlmData2.udiCode].sAlmText;
			tyAlmData2.sRcyMsg	:= a_tyAlmText[tyAlmData2.udiCode].sRcyText;
		END_IF

		sStatTxt	:= tyAlmData2.sAlmMsg;

	ELSIF bRstErr AND (tyAlmData2.udiCode <> 0) THEN

		tyAlmData2.udiCode		:= 0;
		tyAlmData2.eSeverity	:= AlmSeverityNA;
		tyAlmData2.sAlmMsg		:= '';
		tyAlmData2.sRcyMsg		:= '';
		tyAlmData2.bAlm			:= FALSE;
		sStatTxt	:= a_sStatText[eStat];

	END_IF

END_ACTION
```

#### Act_Alarm3.st
```iecst
(** 2020-03-16 **)
ACTION Act_Alarm3:

	//Error
	IF EDGEPOS(eStatus3 = Error) THEN

		tyAlmData3.sProgNm		:= p_sProgNm;
		tyAlmData3.udiCode		:= udiStatus3;
		tyAlmData3.eSeverity	:= AlmSeverityError;
		tyAlmData3.udiRunTime	:= tyAlmData3.udiRunTime + 1;
		tyAlmData3.bAlm			:= TRUE;
		tyAlmData3.udiModuleNum  := udiModuleNum;
		g_sLifterBtmProgNm		:= p_sProgNm;
		//Get Error Message
		IF tyAlmData3.udiCode < 10000 OR tyAlmData3.udiCode > 10299 THEN
			tyAlmData3.sAlmMsg	:= 'Unknown';
			tyAlmData3.sRcyMsg	:= 'Unknown';
		ELSE
			tyAlmData3.sAlmMsg	:= a_tyAlmText[tyAlmData3.udiCode].sAlmText;
			tyAlmData3.sRcyMsg	:= a_tyAlmText[tyAlmData3.udiCode].sRcyText;
		END_IF

		sStatTxt	:= tyAlmData3.sAlmMsg;

	ELSIF bRstErr AND (tyAlmData3.udiCode <> 0) THEN

		tyAlmData3.udiCode		:= 0;
		tyAlmData3.eSeverity	:= AlmSeverityNA;
		tyAlmData3.sAlmMsg		:= '';
		tyAlmData3.sRcyMsg		:= '';
		tyAlmData3.bAlm			:= FALSE;
		sStatTxt	:= a_sStatText[eStat];

	END_IF

END_ACTION
```

#### Act_InitGlobal.st
```iecst
(** 2019-04-09 **)
ACTION Act_InitGlobal:

	(* Always Change If Project Change *)

	//Pass Data To Link
	p_bLinkOpsRun ACCESS p_OpsRun;
	p_bLinkStartupRun ACCESS p_StartupRun;

	p_diLinkSltToSltDist ACCESS p_MagRcpCurrRcpSltToSlt;
	p_bLinkDILifterTimingBeltSen ACCESS p_DILifterTimingBeltSen;
	p_bLinkDILifterSafetyLmtSW1 ACCESS p_DILifterSafetyLmtSW1;
	p_bLinkDILifterSafetyLmtSW2 ACCESS p_DILifterSafetyLmtSW2;

	p_diLinkSltToSltDist1 ACCESS p_MagRcpCurrRcpSltToSlt1;

	p_eLinkMag ACCESS p_NtParamProjMag;
	p_usiLinkMod ACCESS p_ProdRcpCurrRcp1McMod;

	p_diLinkASlt1Pos ACCESS p_MagRcpCurrRcpMag1Slt1Pos;
	p_diLinkBSlt1Pos ACCESS p_MagRcpCurrRcpMag2Slt1Pos;
	p_diLinkCSlt1Pos ACCESS p_MagRcpCurrRcpMag3Slt1Pos;
	p_diLinkDSlt1Pos ACCESS p_MagRcpCurrRcpMag4Slt1Pos;

	p_diLinkASlt1Pos1 ACCESS p_MagRcpCurrRcpMag1Slt1Pos1;
	p_diLinkBSlt1Pos1 ACCESS p_MagRcpCurrRcpMag2Slt1Pos1;
	p_diLinkCSlt1Pos1 ACCESS p_MagRcpCurrRcpMag3Slt1Pos1;
	p_diLinkDSlt1Pos1 ACCESS p_MagRcpCurrRcpMag4Slt1Pos1;

	p_bLinkNtParamProjRotCylPrep ACCESS p_NtParamProjPullerRotCylPrep;

	p_bLinkOpsTravLifULInDSPos ACCESS p_OpsTravLifULInDSPos;

	p_bLinkSafetyRelay ACCESS p_DISafetyRlySig;

	p_bLinkProjLifterMagPlatform ACCESS p_NtParamProjLifterMagPlatform;

	//Pass Data To Internal Use
	p_bEn ACCESS p_DISimServoEn;
	p_udiRstErr ACCESS p_RstErrReset;
	p_bOps ACCESS p_OpsStatusRun;
	p_bManual ACCESS p_UIMnlMod;
//	p_diASlt1Pos ACCESS p_MagRcpCurrRcpMag1Slt1Pos;
//	p_diBSlt1Pos ACCESS p_MagRcpCurrRcpMag2Slt1Pos;
//	p_diCSlt1Pos ACCESS p_MagRcpCurrRcpMag3Slt1Pos;
	p_diAPos ACCESS p_McParamLifterPosA;
	p_diBPos ACCESS p_McParamLifterPosB;
	p_tyTuning ACCESS p_NtParamLifterTuning;
	p_diJogVelInUMPS ACCESS p_UIMnlLifterBtmJogSpd;
	p_diMovePosInUM ACCESS p_UIMnlLifterBtmTargetPos;
	p_diMoveDistInUM ACCESS p_UIMnlLifterBtmStepSize;
	p_bUITeachServo ACCESS p_UITeachServo;
	p_diMoveAcc ACCESS p_NtParamLifterAcc;
	p_diMoveDec ACCESS p_NtParamLifterDec;
	p_bDir ACCESS p_NtParamLifterDir;
	p_usiNode ACCESS p_NtParamLifterNode;
	p_sDevice ACCESS p_NtParamLifterDevice;
	p_sProgNm ACCESS p_NtParamLifterProgNm;
	p_tyParamInHm ACCESS p_NtParamLifterParamInHm;
	p_tyParamInConvert ACCESS p_NtParamLifterParamInConvert;
	p_bNtSettingsLoadDone ACCESS p_StartupNtSettingsLoadDone;
	p_eNtParamMotorType ACCESS p_NtParamLifterMotorType;

	p_bInletShutterCloseRS ACCESS p_DIInShutterCloseRS;
	p_bOutletShutterCloseRS ACCESS p_DIOutShutterCloseRS;
	p_bProjInletShutPrep ACCESS p_NtParamProjInletShutPrep;
	//	p_bInShutterDis ACCESS p_McParamInShutterDis;
	p_bProjOutletShutPrep ACCESS p_NtParamProjOutletShutPrep;
	p_bOutShutterDis ACCESS p_McParamOutShutterDis;
	p_bPullerExtSen ACCESS p_DIPullerExtRS;
	p_bPullerRetSen ACCESS p_DIPullerRetRS;

	p_bDIConvClrSen ACCESS p_DIConvClrSen;
	p_bDIConvLftSen ACCESS p_DIConvLftSen;
	(* Always Change If Project Change *)

END_ACTION
```

#### Act_InitLocal.st
```iecst
(** 2020-03-16 **)
ACTION Act_InitLocal:

	//Input Reference Link To Local Variable
	p_eAct ACCESS ADR(eAct);
	p_udiRstErr ACCESS ADR(udiRstErr);
	p_bPrep ACCESS ADR(bPrep);
	p_bEn ACCESS ADR(bEn);
	p_bDis ACCESS ADR(bDis);
	p_bOps ACCESS ADR(bOps);
	p_bManual ACCESS ADR(bManual);
	p_diGoASlt ACCESS ADR(diGoASlt);
	p_diASltToSltDist ACCESS ADR(diASltToSltDist);
	p_diASlt1Pos ACCESS ADR(diASlt1Pos);
	p_diGoBSlt ACCESS ADR(diGoBSlt);
	p_diBSltToSltDist ACCESS ADR(diBSltToSltDist);
	p_diBSlt1Pos ACCESS ADR(diBSlt1Pos);
	p_diGoCSlt ACCESS ADR(diGoCSlt);
	p_diCSltToSltDist ACCESS ADR(diCSltToSltDist);
	p_diCSlt1Pos ACCESS ADR(diCSlt1Pos);
	p_diGoDSlt ACCESS ADR(diGoDSlt);
	p_diDSltToSltDist ACCESS ADR(diDSltToSltDist);
	p_diDSlt1Pos ACCESS ADR(diDSlt1Pos);
	p_diAPos ACCESS ADR(diAPos);
	p_diBPos ACCESS ADR(diBPos);
	p_diCPos ACCESS ADR(diCPos);
	p_diDPos ACCESS ADR(diDPos);
	p_diEPos ACCESS ADR(diEPos);
	p_diFPos ACCESS ADR(diFPos);
	p_diGPos ACCESS ADR(diGPos);
	p_diHPos ACCESS ADR(diHPos);
	p_tyTuning ACCESS ADR(tyTuning);
	p_diJogVelInUMPS ACCESS ADR(diJogVelInUMPS);
	p_diMovePosInUM ACCESS ADR(diMovePosInUM);
	p_diMoveDistInUM ACCESS ADR(diMoveDistInUM);
	p_diMoveVelInUMPS ACCESS ADR(diMoveVelInUMPS);
	p_diMoveAcc ACCESS ADR(diMoveAcc);
	p_diMoveDec ACCESS ADR(diMoveDec);
	p_diMinAbsPosInUM ACCESS ADR(diMinAbsPosInUM);
	p_diMaxAbsPosInUM ACCESS ADR(diMaxAbsPosInUM);
	p_bInterruptSensor1 ACCESS ADR(bInterruptSensor1);
	p_bInterruptSensor2 ACCESS ADR(bInterruptSensor2);
	p_bInterruptSensor3 ACCESS ADR(bInterruptSensor3);
	p_bInterruptSensor4 ACCESS ADR(bInterruptSensor4);
	p_bInterruptSensor5 ACCESS ADR(bInterruptSensor5);
	p_bInterruptSensor6 ACCESS ADR(bInterruptSensor6);
	p_bDir ACCESS ADR(bDir);
	p_bNoIndexPulse ACCESS ADR(bNoIndexPulse);
	p_usiNode ACCESS ADR(usiNode);
	p_sDevice ACCESS ADR(sDevice);
	p_sProgNm ACCESS ADR(sProgNm);
	p_tyParamInHm ACCESS ADR(tyParamInHm);
	p_tyParamInConvert ACCESS ADR(tyParamInConvert);
	p_bNtSettingsLoadDone ACCESS ADR(bNtSettingsLoadDone);

	p_bInletShutterCloseRS ACCESS ADR(bInletShutterCloseRS);

END_ACTION
```

#### Act_Link.st
```iecst
(** 2019-03-29 **)
ACTION Act_Link:
	IF p_bLinkProjLifterMagPlatform THEN

		p_diASltToSltDist ACCESS p_MagRcpCurrRcpSltToSlt;
		p_diBSltToSltDist ACCESS p_MagRcpCurrRcpSltToSlt;
		p_diCSltToSltDist ACCESS p_MagRcpCurrRcpSltToSlt;
		p_diDSltToSltDist ACCESS p_MagRcpCurrRcpSltToSlt;
	ELSE
		p_diASltToSltDist	:= p_diLinkSltToSltDist * -1;
		p_diBSltToSltDist	:= p_diLinkSltToSltDist * -1;
		p_diCSltToSltDist	:= p_diLinkSltToSltDist * -1;
		p_diDSltToSltDist	:= p_diLinkSltToSltDist * -1;
	END_IF

	p_bInterruptSensor1	:= NOT p_bLinkDILifterTimingBeltSen;
	p_bInterruptSensor2	:= NOT p_bLinkDILifterSafetyLmtSW1;//OR p_bLinkSafetyRelay = FALSE;
	p_bInterruptSensor3	:= NOT p_bLinkDILifterSafetyLmtSW2;

	IF p_bLinkNtParamProjRotCylPrep = FALSE THEN

		IF (p_bProjInletShutPrep = TRUE) AND p_bLinkOpsTravLifULInDSPos = FALSE THEN
			IF p_bInletShutterCloseRS = FALSE OR p_bPullerRetSen = FALSE OR p_bPullerExtSen
				THEN
				p_bInterruptSensor4 := TRUE;
			ELSE
				p_bInterruptSensor4 := FALSE;
			END_IF
		ELSE
			p_bInterruptSensor4 := FALSE;
		END_IF

		IF p_bProjOutletShutPrep = TRUE AND p_bOutShutterDis = FALSE AND p_bLinkOpsTravLifULInDSPos = FALSE THEN
			IF p_bOutletShutterCloseRS = FALSE OR p_bPullerRetSen = FALSE OR p_bPullerExtSen
				THEN
				p_bInterruptSensor5 := TRUE;
			ELSE
				p_bInterruptSensor5 := FALSE;
			END_IF
		ELSE
			p_bInterruptSensor5 := FALSE;
		END_IF

	ELSE

		IF (p_bProjInletShutPrep = TRUE) AND p_bLinkOpsTravLifULInDSPos = FALSE THEN
			IF p_bInletShutterCloseRS = FALSE OR p_bPullerRetSen = FALSE OR p_bPullerExtSen
				THEN
				p_bInterruptSensor4 := TRUE;
			ELSE
				p_bInterruptSensor4 := FALSE;
			END_IF
		ELSE
			p_bInterruptSensor4 := FALSE;
		END_IF

		IF p_bProjOutletShutPrep = TRUE AND p_bOutShutterDis = FALSE AND p_bLinkOpsTravLifULInDSPos = FALSE
			AND p_bLinkProjLifterMagPlatform = FALSE //rotate w/ platform
			THEN
			IF p_bOutletShutterCloseRS = FALSE OR p_bPullerRetSen = FALSE OR p_bPullerExtSen
				THEN
				p_bInterruptSensor5 := TRUE;
			ELSE
				p_bInterruptSensor5 := FALSE;
			END_IF
		ELSE
			p_bInterruptSensor5 := FALSE;
		END_IF
	END_IF

	p_bInterruptSensor6 := (NOT(p_bLinkProjLifterMagPlatform) AND p_bDIConvClrSen) OR p_bDIConvLftSen;

	//p_bDIConvClrSen OR p_bDIConvLftSen;

	IF p_bManual = TRUE THEN
		p_diGoASlt ACCESS p_UIMnlLifterBtmMag1GoSlt;
		p_diGoBSlt ACCESS p_UIMnlLifterBtmMag2GoSlt;
		p_diGoCSlt ACCESS p_UIMnlLifterBtmMag3GoSlt;
		p_diGoDSlt ACCESS p_UIMnlLifterBtmMag4GoSlt;

		p_diMoveVelInUMPS ACCESS p_UIMnlLifterBtmNomSpd;

	ELSE

		IF p_bLinkProjLifterMagPlatform = FALSE THEN
			p_diGoASlt ACCESS p_OpsTravLifLDGoUnloadSlt1;
			p_diGoBSlt ACCESS p_OpsTravLifLDGoUnloadSlt2;
			p_diGoCSlt ACCESS p_OpsTravLifLDGoUnloadSlt3;
			p_diGoDSlt ACCESS p_OpsTravLifLDGoUnloadSlt4;
			p_diMoveVelInUMPS ACCESS p_NtParamLifterAutoSpd;
		ELSE
			p_diGoASlt ACCESS p_OpsLifMagLDGoUnloadSlt1;
			p_diGoBSlt ACCESS p_OpsLifMagLDGoUnloadSlt2;
			p_diGoCSlt ACCESS p_OpsLifMagLDGoUnloadSlt3;
			p_diMoveVelInUMPS ACCESS ADR(diMoveVelInUMPS);
		END_IF

	END_IF

	IF p_eLinkMag = LDMagQuadruple THEN
		CASE p_usiLinkMod OF
			0: //LDModLoadLnA:
				p_diASlt1Pos := p_diLinkASlt1Pos;
				p_diBSlt1Pos := p_diLinkBSlt1Pos;
				p_diCSlt1Pos := p_diLinkCSlt1Pos;
				p_diDSlt1Pos := p_diLinkDSlt1Pos;

				p_diASltToSltDist	:= p_diLinkSltToSltDist * -1;
				p_diBSltToSltDist	:= p_diLinkSltToSltDist * -1;
				p_diCSltToSltDist	:= p_diLinkSltToSltDist * -1;
				p_diDSltToSltDist	:= p_diLinkSltToSltDist * -1;

			1: //LDModLoadLnB:
				p_diASlt1Pos := p_diLinkASlt1Pos1;
				p_diBSlt1Pos := p_diLinkBSlt1Pos1;
				p_diCSlt1Pos := p_diLinkCSlt1Pos1;
				p_diDSlt1Pos := p_diLinkDSlt1Pos1;

				p_diASltToSltDist	:= p_diLinkSltToSltDist1 * -1;
				p_diBSltToSltDist	:= p_diLinkSltToSltDist1 * -1;
				p_diCSltToSltDist	:= p_diLinkSltToSltDist1 * -1;
				p_diDSltToSltDist	:= p_diLinkSltToSltDist1 * -1;

			2: //LDModLoadLnAB:
				p_diASlt1Pos := p_diLinkASlt1Pos;
				p_diBSlt1Pos := p_diLinkBSlt1Pos;
				p_diCSlt1Pos := p_diLinkCSlt1Pos1;
				p_diDSlt1Pos := p_diLinkDSlt1Pos1;

				p_diASltToSltDist	:= p_diLinkSltToSltDist * -1;
				p_diBSltToSltDist	:= p_diLinkSltToSltDist * -1;
				p_diCSltToSltDist	:= p_diLinkSltToSltDist1 * -1;
				p_diDSltToSltDist	:= p_diLinkSltToSltDist1 * -1;
		END_CASE
	ELSE
		p_diASlt1Pos := p_diLinkASlt1Pos;
		p_diBSlt1Pos := p_diLinkBSlt1Pos;
		p_diCSlt1Pos := p_diLinkCSlt1Pos;
		p_diDSlt1Pos := p_diLinkDSlt1Pos;
	END_IF

END_ACTION
```

#### Act_LinkAction.st
```iecst
(** 2019-10-21 **)
ACTION Act_LinkAction:

	IF eStatus = Idle THEN
		IF bModuleNotOK THEN
			p_eAct ACCESS ADR(eAct);
		ELSE
			IF p_bLinkStartupRun = TRUE THEN
				p_eAct ACCESS p_StartupLifterAct;
			ELSIF p_bLinkOpsRun = TRUE THEN
				IF p_bLinkProjLifterMagPlatform  THEN
					p_eAct ACCESS p_OpsLifMagLDLifterAct;
				ELSE
					p_eAct ACCESS p_OpsTravLifLDLifAct;
				END_IF
			ELSIF p_bManual = TRUE THEN
				p_eAct ACCESS p_UILifterBtmAct;
			ELSE
				p_eAct ACCESS ADR(eAct);
			END_IF
		END_IF
	END_IF

	IF EDGENEG(p_bManual) OR EDGENEG(p_bLinkOpsRun) OR EDGENEG(p_bLinkStartupRun) THEN
		tyParamOutDriver.uiCtrlword_6040	:= 0;
	END_IF

END_ACTION
```
